TYPE StackerCranePosition :
STRUCT
	PrePosition	:	REAL;	//Pre-Position for the stacker crane
	Position	:	REAL;	//Position for the stacker crane
END_STRUCT
END_TYPE

(* stored: Version 1.1.0.1
   DUT StackerCranePosition: Id {7ba0fab5-70a2-4a40-8bfa-e03bd55812ab} *)
